// TwinCAT 3 PLC project PLC
// ProgramVersion: 3.1.4023.0
// libraries:
//   Tc2_Standard, * (Beckhoff Automation GmbH)
//   Tc2_System, * (Beckhoff Automation GmbH)
//   Tc3_Module, * (Beckhoff Automation GmbH)
// project tree:
//   / PlcTask.TcTTO
//   POUs/ FB_0221BF00.TcPOU, FB_K50L2.TcPOU, MAIN.TcPOU

CONFIGURATION PLC
    RESOURCE PLC ON TwinCAT3
        TASK PlcTask(INTERVAL := T#10ms, PRIORITY := 20);
        PROGRAM MAIN WITH PlcTask : MAIN;
    END_RESOURCE
END_CONFIGURATION

// ---- POUs/MAIN.TcPOU
PROGRAM MAIN
VAR	
	fbK50L2		 : FB_K50L2;
	fb0221BF00	 : FB_0221BF00;
	
	iCount		: INT;
	tNow		: ULINT := 0;
	tSpace		: ULINT	:= 0;
	tDiff		: ULINT := 100000000;   //TO_ULINT(T#10s);
END_VAR

tNow := F_GetSystemTime();

IF (tNow-tSpace) > tDiff THEN
	tSpace := tNow;
	fb0221BF00(iCount := iCount);
	fbK50L2(iState := iCount);
	iCount := iCount+1;
END_IF

END_PROGRAM

// ---- POUs/FB_K50L2.TcPOU
FUNCTION_BLOCK FB_K50L2
VAR_INPUT
	iState	 : INT;	
END_VAR
VAR
	byOut1	AT %Q* : ARRAY[1..4] OF BYTE;
	//eReadState	: (WAIT,T1,T2,T3);
END_VAR


iState := TO_INT(iState AND TO_INT(16#3));


CASE iState OF
	0:
		byOut1[1] := 16#00;
		byOut1[2] := 16#6;
		byOut1[3] := 16#82;
		byOut1[4] := 16#27;
	1:
		byOut1[1] := 16#00;
		byOut1[2] := 16#1;
		byOut1[3] := 16#88;
		byOut1[4] := 16#2B;
	2:
		byOut1[1] := 16#00;
		byOut1[2] := 16#1;
		byOut1[3] := 16#88;
		byOut1[4] := 16#24;
	3:
		byOut1[1] := 16#00;
		byOut1[2] := 16#4;
		byOut1[3] := 16#88;
		byOut1[4] := 16#22;
END_CASE

END_FUNCTION_BLOCK

// ---- POUs/FB_0221BF00.TcPOU
FUNCTION_BLOCK FB_0221BF00
VAR_INPUT
	iCount	 : INT;	
END_VAR
VAR
	byB1  AT%Q*	: BOOL;
	byB2  AT%Q*	: BOOL;
	byB3  AT%Q*	: BOOL;
	byB4  AT%Q*	: BOOL;
	byB5  AT%Q*	: BOOL;
	byB6  AT%Q*	: BOOL;
	byB7  AT%Q*	: BOOL;
	byB8  AT%Q*	: BOOL;
END_VAR

	byB1 	:= iCount.0;
	byB2	:= iCount.1;
	byB3	:= iCount.2;
	byB4 	:= iCount.3;
	byB5	:= iCount.4;
	byB6	:= iCount.5;
	byB7	:= iCount.6;
	byB8	:= iCount.7;

END_FUNCTION_BLOCK
